PROGRAM main
VAR
	CountPulse AT %QX0.0 : bool;
	ResetCounter AT %QX0.1 : bool;
	Done AT %QX0.2 : bool;
	CounterEnabled AT %QX0.3 : bool;
	Overflow AT %QX0.4 : bool;
	CurrentCount AT %MD0 : dint;
	CounterInstance : TF_CTU;
	Preset : dint := 3;
END_VAR

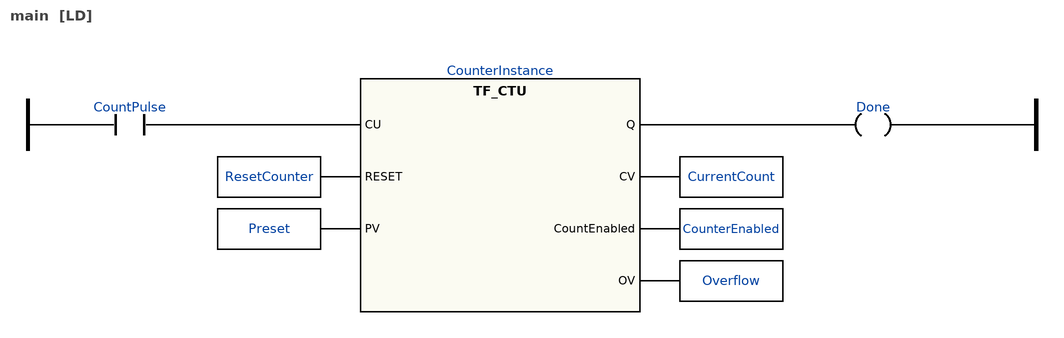
(* LD diagram, written out as Structured Text *)
CounterInstance(CU := CountPulse, RESET := ResetCounter, PV := Preset);
Done := CounterInstance.Q;
CurrentCount := CounterInstance.CV;
CounterEnabled := CounterInstance.CountEnabled;
Overflow := CounterInstance.OV;
END_PROGRAM
